// TIA Portal V16 export
// export: Created 2022-07-21T09:35:16.6422046Z, ExportSetting WithDefaults, DisplayName Totally Integrated Automation Portal, DisplayVersion V16 Update 4, DisplayName TIA Portal Version Control Interface, DisplayVersion V16 Update 2, DisplayName TIA Portal Openness, DisplayVersion V16 Update 4, DisplayName SINAMICS Startdrive Advanced, DisplayVersion V16 Update 5, DisplayName SINAMICS Startdrive G130, G150, S120, S150, SINAMICS MV, S210, DisplayVersion V16 Update 5, DisplayName SINAMICS Startdrive G110M, G120, G120C, G120D, G120P, G115D, DisplayVersion V16 Update 5, DisplayName STEP 7 Professional, DisplayVersion V16 Update 4, DisplayName STEP 7 Safety, DisplayVersion V16, DisplayName WinCC Advanced, DisplayVersion V16 Update 4
FUNCTION_BLOCK "fbMessageError"   // FB118, LAD
TITLE = Error handling / Obsługa błędów
{ S7_Optimized_Access := 'TRUE' }
VERSION : 0.1
// stored: AutoNumber true, IsIECCheckEnabled true, IsRetainMemResEnabled false, MemoryReserve 100, SetENOAutomatically false, UDAEnableTagReadback false
   VAR_INPUT
      inEnable { ExternalAccessible := 'False'; ExternalVisible := 'False'; ExternalWritable := 'False'} : Bool;   // Zezwolenie / Enable
      inFbSignalOk { ExternalAccessible := 'False'; ExternalVisible := 'False'; ExternalWritable := 'False'} : Bool;   // Sygnał ok / Signal ok
      inResetMessages { ExternalAccessible := 'False'; ExternalVisible := 'False'; ExternalWritable := 'False'} : Bool;   // Reset
      inDelaySignalOn { ExternalAccessible := 'False'; ExternalVisible := 'False'; ExternalWritable := 'False'} : Time;   // Opóźnienie załączenia / on delay
      inDelaySignalOff { ExternalAccessible := 'False'; ExternalVisible := 'False'; ExternalWritable := 'False'} : Time;   // Opóźnienie wyłączenia / off delay
   END_VAR
   VAR_OUTPUT
      ouMessage { ExternalAccessible := 'False'; ExternalVisible := 'False'; ExternalWritable := 'False'} : Bool;   // Sygnał wyjściowy [1 - błąd] / error output
   END_VAR
   VAR
      sMessage { ExternalAccessible := 'False'; ExternalVisible := 'False'; ExternalWritable := 'False'; S7_SetPoint := 'True'} : "fbMessageHandlingDelayed";
   END_VAR
BEGIN

REGION Network 1: Call error handling / Wywołanie bloczka do błędu
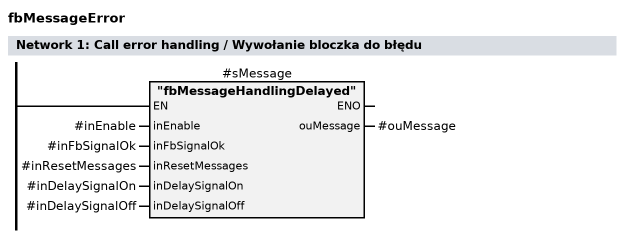
   RUNG wire#powerrail
      #sMessage(inEnable := #inEnable, inFbSignalOk := #inFbSignalOk, inResetMessages := #inResetMessages, inDelaySignalOn := #inDelaySignalOn, inDelaySignalOff := #inDelaySignalOff, ouMessage => #ouMessage)
   END_RUNG
   // the same network as SCL:
   #sMessage(inEnable := #inEnable,   // "fbMessageHandlingDelayed"
             inFbSignalOk := #inFbSignalOk,
             inResetMessages := #inResetMessages,
             inDelaySignalOn := #inDelaySignalOn,
             inDelaySignalOff := #inDelaySignalOff,
             ouMessage => #ouMessage);
END_REGION
END_FUNCTION_BLOCK
